// TIA Portal V19 export
TYPE "Positioning_MOL_Machine_Wng"
// stored: Access Published
   STRUCT
      NotAutReady : Bool;   // Machine NOT Ready for automatic start
      Minus_CndMissing : Bool;   // Lack of conditions for movement in negative direction
      Plus_CndMissing : Bool;   // Lack of conditions for movement in positive direction
      Ax_NotHomed : Bool;   // Axis not homed / referenced
      Ax : "OOAx_Wng";   // ON-OFF AXIS
   END_STRUCT;
   // // Ax.SwLimitMinus : Negative software limit reached / exceeded.
   // // Ax.SwLimitPlus : Positive software limit reached / exceeded.
END_TYPE
